//La FB1 Implementa l'interfaccia iFB

FUNCTION_BLOCK PUBLIC FB1 IMPLEMENTS iFb
VAR_INPUT
END_VAR
VAR_OUTPUT
END_VAR
VAR
	fInternalInput1 : REAL;
	fInternalInput2 : REAL;
END_VAR

;

{warning 'add property implementation'}
PROPERTY fInput1 : REAL
GET
fInput1 := this^.fInternalInput1;
END_GET
SET
this^.fInternalInput1 := fInput1;
END_SET
END_PROPERTY

{warning 'add property implementation'}
PROPERTY fInput2 : REAL
GET
fInput2 := this^.fInternalInput2;
END_GET
SET
this^.fInternalInput2 := fInput2;
END_SET
END_PROPERTY

{warning 'add method implementation'}
METHOD returnValue : REAL
//Implementazione Interfaccia con somma
returnValue := this^.fInput1 + this^.fInput2;
END_METHOD

END_FUNCTION_BLOCK

(* stored: Version 1.1.0.1, ProductVersion 3.1.4022.16
   POU FB1: Id {06b68a36-e277-4926-ba89-7478bf46f8c0}, SpecialFunc None
   Property fInput1: Id {df74346d-8b45-4c32-ac3d-33428ff8fec5}
   Get Get: Id {69ac556e-135e-4c2f-a6a9-ab463f701730}
   Set Set: Id {1fbc8862-20fd-429f-b0af-6e53f24b57d7}
   Property fInput2: Id {26ca5f64-78c4-45d8-8019-f1a3ec9fc7f1}
   Get Get: Id {c29ad947-b7f8-4ea7-bc5e-0c930aa5b530}
   Set Set: Id {2d912acc-3279-46a3-83af-16d4bdb35004}
   Method returnValue: Id {09bb01fa-c323-4a0a-a317-12d6398f3bc8} *)
